FUNCTION_BLOCK MyApplInterface
  (* Version 01.00, 2002-12-12, Updated with Status output *)
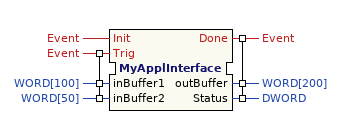
  EVENT_INPUT
    Init;
    Trig WITH inBuffer1, inBuffer2;
  END_EVENT
  EVENT_OUTPUT
    Done WITH outBuffer, Status;
  END_EVENT
  VAR_INPUT
    inBuffer1 : ARRAY [0..99] OF WORD;
    inBuffer2 : ARRAY [0..49] OF WORD;
  END_VAR
  VAR_OUTPUT
    outBuffer : ARRAY [0..199] OF WORD;
    Status : DWORD;
  END_VAR
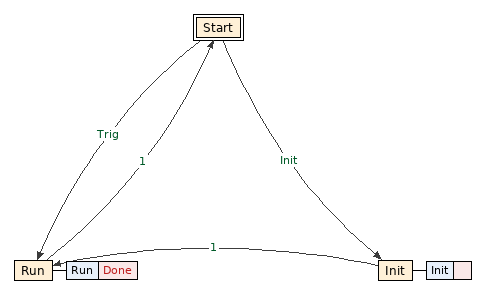
  EC_STATES
    Start;
    Init : Init;
    Run : Run -> Done;
  END_STATES
  EC_TRANSITIONS
    Start TO Init := Init;
    Init TO Run := 1;
    Start TO Run := Trig;
    Run TO Start := 1;
  END_TRANSITIONS
  ALGORITHM Init IN ST:

  END_ALGORITHM
  ALGORITHM Run IN ST:

  END_ALGORITHM
END_FUNCTION_BLOCK
